TYPE T_Ctrl_SIf_LAI_Cfg :
STRUCT
END_STRUCT
END_TYPE

(* stored: Version 1.1.0.1, ProductVersion 3.1.0.19
   DUT T_Ctrl_SIf_LAI_Cfg: Id {1bec4058-e50a-481d-8eba-88bfcb4e93bd} *)
